Fanuc KAREL source: kt00146.compact.KL

PROGRAM KT00146
%STACKSIZE=65535
%PRIORITY=65535
%NOLOCKGROUP
VAR
Y1 : ARRAY[2] OF BYTE
I2 : INTEGER
OUT : REAL
BEGIN
Y1[1]=2
I2=3
OUT=((Y1[1] DIV I2))
END KT00146
